TYPE DUT_SKILL_INPUT :
STRUCT
	///Range of parameters
	ParameterInput: ARRAY[0..ParameterCnt] OF DUT_PARAMETER_INPUT;
	///Start process
	Execute: BOOL;
END_STRUCT
END_TYPE

(* stored: Version 1.1.0.1, ProductVersion 3.1.0.25
   DUT DUT_SKILL_INPUT: Id {e21748c8-497f-48ae-90e6-9d7e80104bf5} *)
